// TIA Portal project "Brock_wyklad" (V17)

(* hardware
DEVICE "S7-1500/ET200MP station_1"  S7-1500 station
   slot 0: "Rail_0"  Rack  6ES7 590-1***0-0AA0
   slot 1: "PLC_1"  CPU 1515-2 PN  6ES7 515-2AM02-0AB0  V2.9
      slot 3: "CPU display_1"  6ES7591-1BA00-0AA0
      slot 32768: "PROFINET interface_1"  X1
         slot 32769: "Port_1"  X1 P1
         slot 32770: "Port_2"  X1 P2
      slot 33024: "PROFINET interface_2"  X2
         slot 33025: "Port_1"  X2 P1
      slot 34817: "Virtual CP interface port_1"  Virtual CP interface port  Virtual CP interface port
*)

// ===== PLC "PLC_1"  CPU 1515-2 PN =====

DATA_BLOCK "Swiatla_DB"   // DB1
{ S7_Optimized_Access := 'TRUE' }
VERSION : 0.1
   VAR
      reset : Bool := true;
      czujnik1 : Bool;
      czujnik2 : Bool;
      czujnik3 : Bool;
      out0 : Bool;
      out1 : Bool;
      out2 : Bool;
      out3 : Bool;
      out4 : Bool;
      out5 : Bool;
      m1 : Bool;
      m2 : Bool;
      m3 : Bool;
      m4 : Bool;
      m5 : Bool;
   END_VAR
BEGIN
END_DATA_BLOCK

DATA_BLOCK "Swiatla_sekwencja_DB"   // DB2
{ S7_Optimized_Access := 'TRUE' }
VERSION : 0.1
// stored: InstanceOfName Swiatla_sekwencja
"Swiatla_sekwencja"
BEGIN
END_DATA_BLOCK

DATA_BLOCK "Swiatla_LAD_DB"   // DB7
{ S7_Optimized_Access := 'TRUE' }
VERSION : 0.1
// stored: InstanceOfName Swiatla_LAD
"Swiatla_LAD"
BEGIN
END_DATA_BLOCK

// folder: System blocks/Program resources

DATA_BLOCK "IEC_Timer_0_DB"   // DB3
{ S7_Optimized_Access := 'TRUE' }
AUTHOR : Simatic
FAMILY : IEC
NAME : IEC_TMR
VERSION : 1.0
// stored: InstanceOfName IEC_TIMER
"IEC_TIMER"
BEGIN
END_DATA_BLOCK

DATA_BLOCK "IEC_Timer_1_DB"   // DB4
{ S7_Optimized_Access := 'TRUE' }
AUTHOR : Simatic
FAMILY : IEC
NAME : IEC_TMR
VERSION : 1.0
// stored: InstanceOfName IEC_TIMER
"IEC_TIMER"
BEGIN
END_DATA_BLOCK

DATA_BLOCK "IEC_Timer_2_DB"   // DB5
{ S7_Optimized_Access := 'TRUE' }
AUTHOR : Simatic
FAMILY : IEC
NAME : IEC_TMR
VERSION : 1.0
// stored: InstanceOfName IEC_TIMER
"IEC_TIMER"
BEGIN
END_DATA_BLOCK

DATA_BLOCK "IEC_Timer_3_DB"   // DB6
{ S7_Optimized_Access := 'TRUE' }
AUTHOR : Simatic
FAMILY : IEC
NAME : IEC_TMR
VERSION : 1.0
// stored: InstanceOfName IEC_TIMER
"IEC_TIMER"
BEGIN
END_DATA_BLOCK

// folder: (top level)

FUNCTION_BLOCK "Swiatla_sekwencja"   // FB1, GRAPH_PLUS
{ S7_Optimized_Access := 'TRUE' }
VERSION : 0.1
   VAR_INPUT
      OFF_SQ : Bool := false;   // Turn sequence off
      INIT_SQ : Bool := false;   // Set sequence to initial state
      ACK_EF : Bool := false;   // Acknowledge all errors and faults
      S_PREV : Bool := false;   // Output previous step in parameter S_NO
      S_NEXT : Bool := false;   // Indicate next step in parameter S_NO
      SW_AUTO : Bool := false;   // Automatic mode
      SW_TAP : Bool := false;   // Semiautomatic/switch with transition
      SW_TOP : Bool := false;   // Semiautomatic/ignore transition
      SW_MAN : Bool := false;   // Manual mode
      S_SEL : Int := 0;   // Select step to be output to S_NO
      S_ON : Bool := false;   // Activate step indicated in S_NO
      S_OFF : Bool := false;   // Deactivate step indicated S_NO
      T_PUSH : Bool := false;   // Enable transition to switch in semi automatic mode
   END_VAR
   VAR_OUTPUT
      S_NO : Int := 0;   // Step number
      S_MORE : Bool := false;   // More steps are available and can be shown in S_NO
      S_ACTIVE : Bool := false;   // Step indicated in S_NO is active
      ERR_FLT : Bool := false;   // Interlock or supervision group error
      AUTO_ON : Bool := false;   // Automatic mode is active
      TAP_ON : Bool := false;   // Semiautomatic mode/step with transition enabled
      TOP_ON : Bool := false;   // Semiautomatic mode/ignore transition enabled
      MAN_ON : Bool := false;   // Manual mode is active
   END_VAR
   VAR
      HMI_INFO : Array[0..8] of UInt;
      IF_PAR : G7_IfParPlus_V6;
      RT_DATA : G7_RTDataPlus_V6;   // Internal data area
      "I0 and I1 positive" : G7_TransitionPlus_V6;   // Transition structure
      Trans2 : G7_TransitionPlus_V6;   // Transition structure
      Trans3 : G7_TransitionPlus_V6;   // Transition structure
      Trans4 : G7_TransitionPlus_V6;   // Transition structure
      Trans5 : G7_TransitionPlus_V6;   // Transition structure
      Trans6 : G7_TransitionPlus_V6;   // Transition structure
      Trans7 : G7_TransitionPlus_V6;   // Transition structure
      Trans9 : G7_TransitionPlus_V6;   // Transition structure
      Trans10 : G7_TransitionPlus_V6;   // Transition structure
      Trans11 : G7_TransitionPlus_V6;   // Transition structure
      Trans12 : G7_TransitionPlus_V6;   // Transition structure
      Step1 : G7_StepPlus_V6;   // Step structure
      Step2 : G7_StepPlus_V6;   // Step structure
      Step3 : G7_StepPlus_V6;   // Step structure
      Step4 : G7_StepPlus_V6;   // Step structure
      "Positive edge I1" : G7_StepPlus_V6;   // Step structure
      Step6 : G7_StepPlus_V6;   // Step structure
      Step7 : G7_StepPlus_V6;   // Step structure
      SINI : Array[0..1] of USInt;
      LSTT : Array[0..10] of USInt;
      ATAJ : Array[0..10] of USInt;
      ATAB : Array[0..10] of USInt;
      PSTT : Array[0..10] of USInt;
      NSTT : Array[0..10] of USInt;
      ASSJ : Array[0..6] of USInt;
      ASSB : Array[0..6] of USInt;
      PTTS : Array[0..6] of USInt;
      NTTS : Array[0..6] of USInt;
      SW_SQTS : Array[0..6] of USInt;
      SWITCH : Array[0..3] of USInt;
      TVX : Array[0..9] of USInt;
      TTX : Array[0..9] of USInt;
      TSX : Array[0..1] of USInt;
      S00X : Array[0..1] of USInt;
      SOFFX : Array[0..1] of USInt;
      SONX : Array[0..1] of USInt;
      SAX : Array[0..1] of USInt;
      SERRX : Array[0..7] of USInt;
      SMX : Array[0..7] of USInt;
      S0X : Array[0..7] of USInt;
      S1X : Array[0..7] of USInt;
      IL_ALARM_INST : Diag_Alarm;
      SUP_ALARM_INST : Diag_Alarm;
      STEP_TIME_ALARM_INST : Diag_Alarm;
      IEC_TIMER_INST : IEC_TIMER;
      TRANSACTION_FLAG : Bool := false;
   END_VAR
   // SINI[0] := 2;
   // LSTT[0] := 255;
   // LSTT[1] := 255;
   // LSTT[2] := 255;
   // LSTT[3] := 255;
   // LSTT[4] := 255;
   // LSTT[5] := 255;
   // ATAJ[1] := 1;
   // ATAJ[2] := 2;
   // ATAJ[3] := 3;
   // ATAJ[4] := 4;
   // ATAJ[5] := 5;
   // ATAJ[6] := 6;
   // ATAB[1] := 7;
   // ATAB[2] := 8;
   // ATAB[3] := 9;
   // ATAB[4] := 4;
   // ATAB[5] := 10;
   // ATAB[6] := 6;
   // PSTT[1] := 1;
   // PSTT[2] := 2;
   // PSTT[3] := 3;
   // PSTT[4] := 4;
   // PSTT[5] := 5;
   // PSTT[6] := 6;
   // NSTT[0] := 4;
   // NSTT[1] := 2;
   // NSTT[2] := 3;
   // NSTT[3] := 5;
   // NSTT[4] := 1;
   // NSTT[5] := 6;
   // ASSJ[1] := 1;
   // ASSJ[2] := 2;
   // ASSJ[3] := 3;
   // ASSJ[4] := 4;
   // ASSJ[5] := 5;
   // ASSJ[6] := 6;
   // ASSB[1] := 1;
   // ASSB[2] := 2;
   // ASSB[3] := 3;
   // ASSB[4] := 4;
   // ASSB[5] := 5;
   // ASSB[6] := 6;
   // PTTS[0] := 255;
   // PTTS[1] := 4;
   // PTTS[2] := 1;
   // PTTS[3] := 2;
   // PTTS[5] := 3;
   // PTTS[6] := 5;
   // NTTS[1] := 1;
   // NTTS[2] := 2;
   // NTTS[3] := 3;
   // NTTS[4] := 4;
   // NTTS[5] := 5;
   // NTTS[6] := 6;
   // TVX[0] := 16#1;
   // TTX[0] := 16#1;
   // TSX[0] := 16#1;
   // S00X[0] := 16#1;
   // SOFFX[0] := 16#1;
   // SONX[0] := 16#1;
   // SAX[0] := 16#1;
   // SERRX[0] := 16#1;
   // SMX[0] := 16#1;
   // S0X[0] := 16#1;
   // S1X[0] := 16#1;
   // ATAJ[7] := 7;
   // ATAJ[8] := 8;
   // ATAJ[9] := 9;
   // ATAJ[10] := 10;
   // ATAB[7] := 1;
   // ATAB[8] := 2;
   // ATAB[9] := 3;
   // ATAB[10] := 5;
   // PSTT[7] := 1;
   // PSTT[8] := 2;
   // PSTT[9] := 3;
   // PSTT[10] := 5;
   // SW_SQTS[2] := 1;
   // SW_SQTS[3] := 2;
   // SW_SQTS[5] := 3;
   // SW_SQTS[6] := 4;
BEGIN
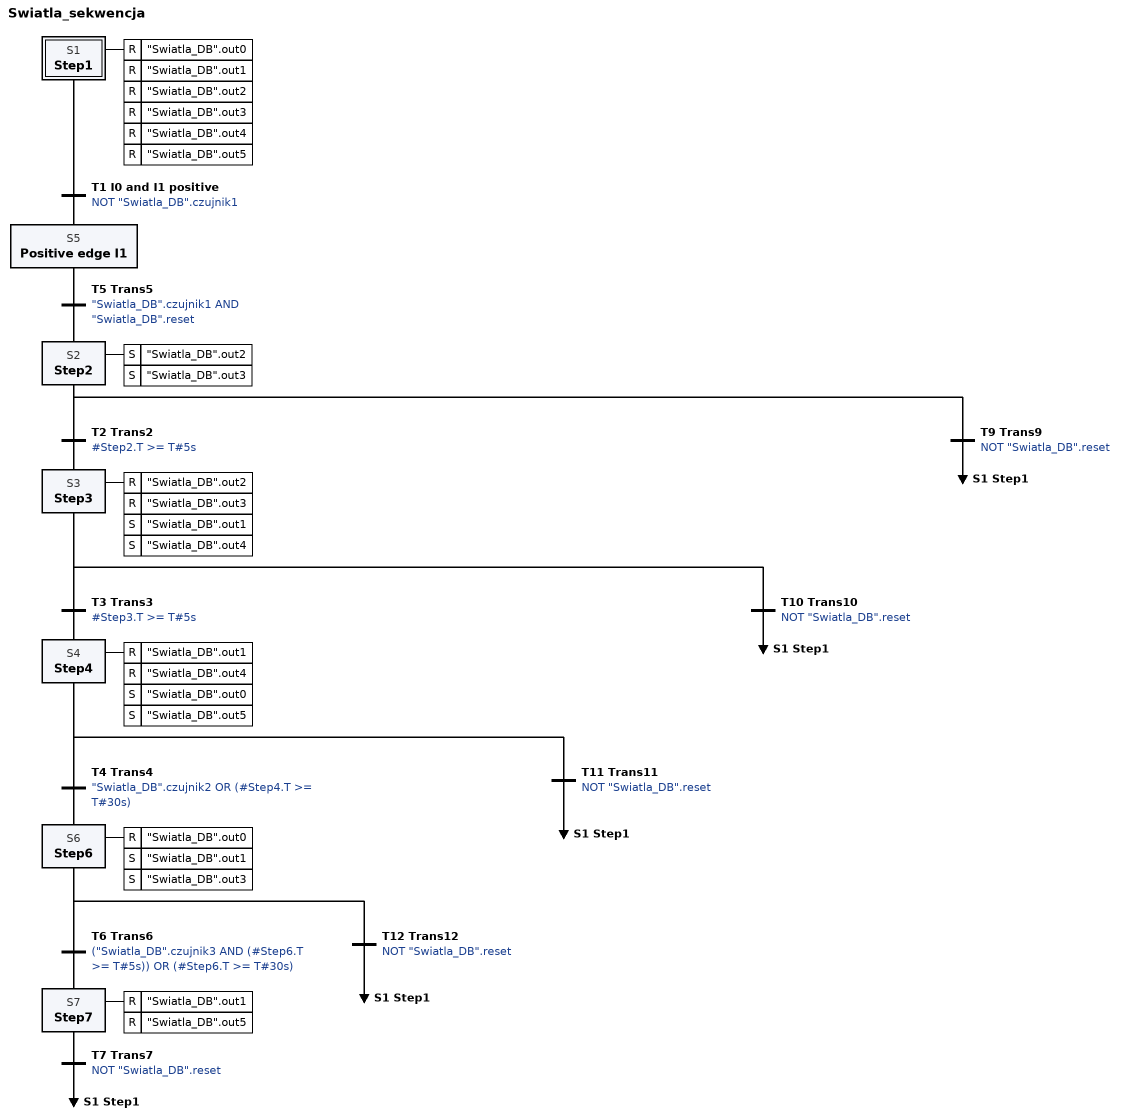
   // sequencer 1
   INITIAL_STEP Step1:   // S1, max time T#10S, warning time T#7S
              R    "Swiatla_DB".out0
              R    "Swiatla_DB".out1
              R    "Swiatla_DB".out2
              R    "Swiatla_DB".out3
              R    "Swiatla_DB".out4
              R    "Swiatla_DB".out5
   END_STEP
   TRANSITION "I0 and I1 positive" FROM Step1 TO "Positive edge I1"   // T1
      := NOT "Swiatla_DB".czujnik1;
   END_TRANSITION
   STEP Step2:   // S2, max time T#10S, warning time T#7S
              S    "Swiatla_DB".out2
              S    "Swiatla_DB".out3
   END_STEP
   TRANSITION Trans2 FROM Step2 TO Step3   // T2
      := #Step2.T >= T#5s;
   END_TRANSITION
   TRANSITION Trans9 FROM Step2 TO Step1   // T9, jump
      := NOT "Swiatla_DB".reset;
   END_TRANSITION
   STEP Step3:   // S3, max time T#10S, warning time T#7S
              R    "Swiatla_DB".out2
              R    "Swiatla_DB".out3
              S    "Swiatla_DB".out1
              S    "Swiatla_DB".out4
   END_STEP
   TRANSITION Trans3 FROM Step3 TO Step4   // T3
      := #Step3.T >= T#5s;
   END_TRANSITION
   TRANSITION Trans10 FROM Step3 TO Step1   // T10, jump
      := NOT "Swiatla_DB".reset;
   END_TRANSITION
   STEP Step4:   // S4, max time T#10S, warning time T#7S
              R    "Swiatla_DB".out1
              R    "Swiatla_DB".out4
              S    "Swiatla_DB".out0
              S    "Swiatla_DB".out5
   END_STEP
   TRANSITION Trans4 FROM Step4 TO Step6   // T4
      := "Swiatla_DB".czujnik2 OR (#Step4.T >= T#30s);
   END_TRANSITION
   TRANSITION Trans11 FROM Step4 TO Step1   // T11, jump
      := NOT "Swiatla_DB".reset;
   END_TRANSITION
   STEP "Positive edge I1":   // S5, max time T#10S, warning time T#7S
   END_STEP
   TRANSITION Trans5 FROM "Positive edge I1" TO Step2   // T5
      := "Swiatla_DB".czujnik1 AND "Swiatla_DB".reset;
   END_TRANSITION
   STEP Step6:   // S6, max time T#10S, warning time T#7S
              R    "Swiatla_DB".out0
              S    "Swiatla_DB".out1
              S    "Swiatla_DB".out3
   END_STEP
   TRANSITION Trans6 FROM Step6 TO Step7   // T6
      := ("Swiatla_DB".czujnik3 AND (#Step6.T >= T#5s)) OR (#Step6.T >= T#30s);
   END_TRANSITION
   TRANSITION Trans12 FROM Step6 TO Step1   // T12, jump
      := NOT "Swiatla_DB".reset;
   END_TRANSITION
   STEP Step7:   // S7, max time T#10S, warning time T#7S
              R    "Swiatla_DB".out1
              R    "Swiatla_DB".out5
   END_STEP
   TRANSITION Trans7 FROM Step7 TO Step1   // T7, jump
      := NOT "Swiatla_DB".reset;
   END_TRANSITION
END_FUNCTION_BLOCK

FUNCTION_BLOCK "Swiatla_LAD"   // FB2, LAD
{ S7_Optimized_Access := 'TRUE' }
VERSION : 0.1
   VAR_INPUT
      I0 : Bool;
      I1 : Bool;
      I2 : Bool;
      I3 : Bool;
   END_VAR
   VAR_OUTPUT
      out0 : Bool;
      out1 : Bool;
      out2 : Bool;
      out3 : Bool;
      out4 : Bool;
      out5 : Bool;
   END_VAR
   VAR_IN_OUT
      M1 : Bool;
      M2 : Bool;
      M3 : Bool;
      M4 : Bool;
      M5 : Bool;
   END_VAR
   VAR
      M0 : Bool;
      I1_static : Bool;
   END_VAR
   VAR_TEMP   // added for the SCL form of the ladder/FBD networks
      _w1 : Bool;
   END_VAR
BEGIN

REGION Network 1
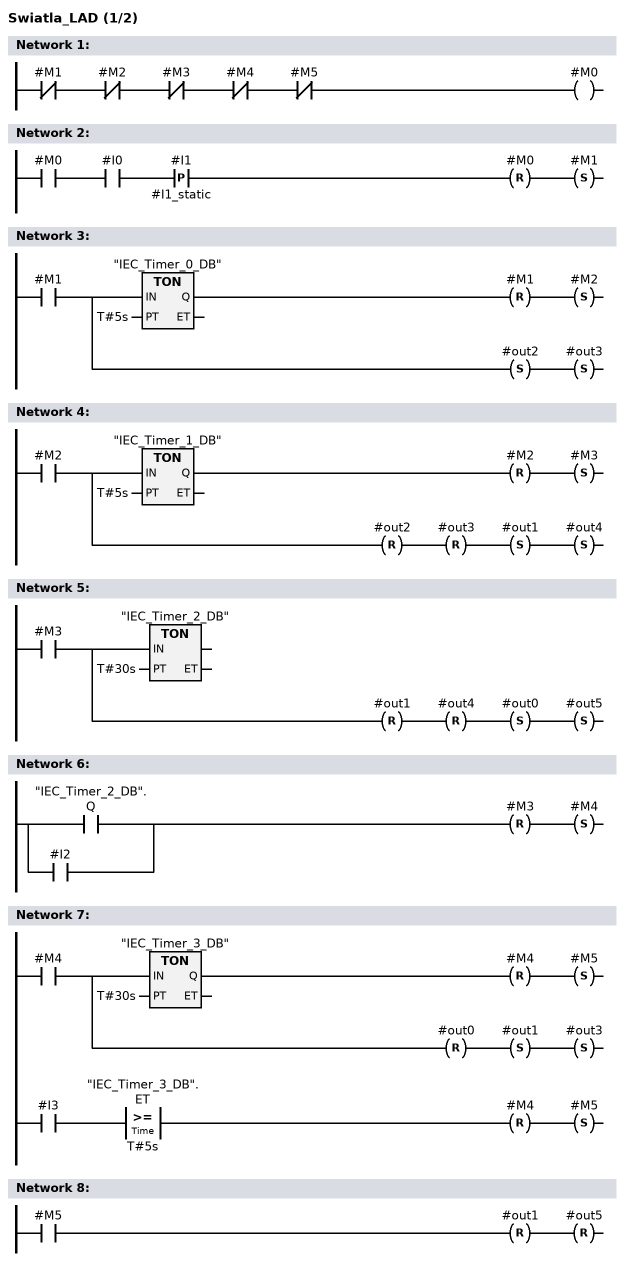
   RUNG wire#powerrail
      I_Contact( #M1 )
      I_Contact( #M2 )
      I_Contact( #M3 )
      I_Contact( #M4 )
      I_Contact( #M5 )
      Coil( #M0 )
   END_RUNG
   // the same network as SCL:
   #M0 := NOT #M1 AND NOT #M2 AND NOT #M3 AND NOT #M4 AND NOT #M5;
END_REGION

REGION Network 2
   RUNG wire#powerrail
      Contact( #M0 )
      Contact( #I0 )
      P_Contact(operand := #I1, bit := #I1_static)
      R_Coil( #M0 )
      S_Coil( #M1 )
   END_RUNG
   // the same network as SCL:
   #_w1 := #M0 AND #I0 AND #I1 AND NOT #I1_static;   // rising edge of #I1
   #I1_static := #I1;
   IF #_w1 THEN
       #M0 := FALSE;
       #M1 := TRUE;
   END_IF;
END_REGION

REGION Network 3
   "IEC_Timer_0_DB".TON(IN := #M1, PT := T#5s);
   #_w1 := #M1;
   IF "IEC_Timer_0_DB".Q THEN
       #M1 := FALSE;
       #M2 := TRUE;
   END_IF;
   IF #_w1 THEN
       #out2 := TRUE;
       #out3 := TRUE;
   END_IF;
END_REGION

REGION Network 4
   "IEC_Timer_1_DB".TON(IN := #M2, PT := T#5s);
   #_w1 := #M2;
   IF "IEC_Timer_1_DB".Q THEN
       #M2 := FALSE;
       #M3 := TRUE;
   END_IF;
   IF #_w1 THEN
       #out2 := FALSE;
       #out3 := FALSE;
       #out1 := TRUE;
       #out4 := TRUE;
   END_IF;
END_REGION

REGION Network 5
   "IEC_Timer_2_DB".TON(IN := #M3, PT := T#30s);
   IF #M3 THEN
       #out1 := FALSE;
       #out4 := FALSE;
       #out0 := TRUE;
       #out5 := TRUE;
   END_IF;
END_REGION

REGION Network 6
   RUNG wire#powerrail
      Contact( "IEC_Timer_2_DB".Q )
      wire#w1
      R_Coil( #M3 )
      S_Coil( #M4 )
   END_RUNG
   RUNG wire#powerrail
      Contact( #I2 )
   END_RUNG wire#w1
   // the same network as SCL:
   IF "IEC_Timer_2_DB".Q OR #I2 THEN
       #M3 := FALSE;
       #M4 := TRUE;
   END_IF;
END_REGION

REGION Network 7
   "IEC_Timer_3_DB".TON(IN := #M4, PT := T#30s);
   #_w1 := #M4;
   IF "IEC_Timer_3_DB".Q THEN
       #M4 := FALSE;
       #M5 := TRUE;
   END_IF;
   IF #_w1 THEN
       #out0 := FALSE;
       #out1 := TRUE;
       #out3 := TRUE;
   END_IF;
   IF #I3 AND ("IEC_Timer_3_DB".ET >= T#5s) THEN
       #M4 := FALSE;
       #M5 := TRUE;
   END_IF;
END_REGION

REGION Network 8
   RUNG wire#powerrail
      Contact( #M5 )
      R_Coil( #out1 )
      R_Coil( #out5 )
   END_RUNG
   // the same network as SCL:
   IF #M5 THEN
       #out1 := FALSE;
       #out5 := FALSE;
   END_IF;
END_REGION

REGION Network 9
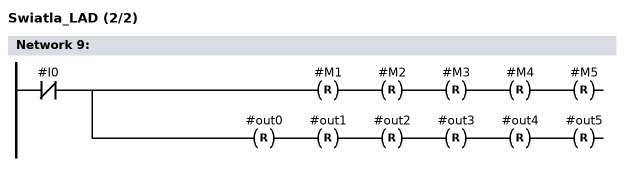
   RUNG wire#powerrail
      I_Contact( #I0 )
      wire#w1
      R_Coil( #M1 )
      R_Coil( #M2 )
      R_Coil( #M3 )
      R_Coil( #M4 )
      R_Coil( #M5 )
   END_RUNG
   RUNG wire#w1
      R_Coil( #out0 )
      R_Coil( #out1 )
      R_Coil( #out2 )
      R_Coil( #out3 )
      R_Coil( #out4 )
      R_Coil( #out5 )
   END_RUNG
   // the same network as SCL:
   IF NOT #I0 THEN
       #M1 := FALSE;
       #M2 := FALSE;
       #M3 := FALSE;
       #M4 := FALSE;
       #M5 := FALSE;
       #out0 := FALSE;
       #out1 := FALSE;
       #out2 := FALSE;
       #out3 := FALSE;
       #out4 := FALSE;
       #out5 := FALSE;
   END_IF;
END_REGION
END_FUNCTION_BLOCK

ORGANIZATION_BLOCK "Main"   // OB1, LAD, ProgramCycle
TITLE = "Main Program Sweep (Cycle)"
{ S7_Optimized_Access := 'TRUE' }
VERSION : 0.1
   VAR_INPUT
      Initial_Call : Bool;   // Initial call of this OB
      Remanence : Bool;   // =True, if remanent data are available
   END_VAR
BEGIN

REGION Network 1
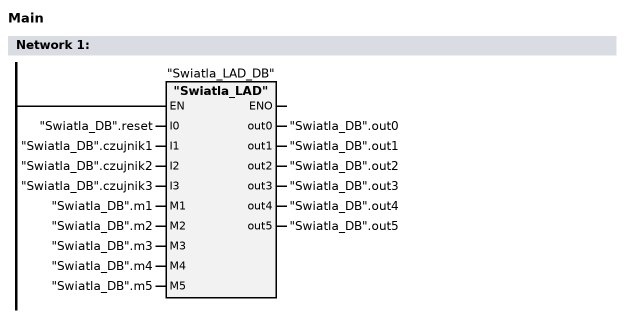
   RUNG wire#powerrail
      "Swiatla_LAD_DB"(I0 := "Swiatla_DB".reset, I1 := "Swiatla_DB".czujnik1, I2 := "Swiatla_DB".czujnik2, I3 := "Swiatla_DB".czujnik3, M1 := "Swiatla_DB".m1, M2 := "Swiatla_DB".m2, M3 := "Swiatla_DB".m3, M4 := "Swiatla_DB".m4, M5 := "Swiatla_DB".m5, out0 => "Swiatla_DB".out0, out1 => "Swiatla_DB".out1, out2 => "Swiatla_DB".out2, out3 => "Swiatla_DB".out3, out4 => "Swiatla_DB".out4, out5 => "Swiatla_DB".out5)
   END_RUNG
   // the same network as SCL:
   "Swiatla_LAD_DB"(I0 := "Swiatla_DB".reset,   // "Swiatla_LAD"
                    I1 := "Swiatla_DB".czujnik1,
                    I2 := "Swiatla_DB".czujnik2,
                    I3 := "Swiatla_DB".czujnik3,
                    M1 := "Swiatla_DB".m1,
                    M2 := "Swiatla_DB".m2,
                    M3 := "Swiatla_DB".m3,
                    M4 := "Swiatla_DB".m4,
                    M5 := "Swiatla_DB".m5,
                    out0 => "Swiatla_DB".out0,
                    out1 => "Swiatla_DB".out1,
                    out2 => "Swiatla_DB".out2,
                    out3 => "Swiatla_DB".out3,
                    out4 => "Swiatla_DB".out4,
                    out5 => "Swiatla_DB".out5);
END_REGION
END_ORGANIZATION_BLOCK